// TIA Portal V19 export
FUNCTION_BLOCK "EXCHANGETRAY_ConstraintRollerCmResetOperator"   // FB51, LAD
TITLE = description
// REGION BLOCK INFO HEADER
//     //===============================================================================
//     // (company)/ (c)Copyright (year)
//     //-------------------------------------------------------------------------------
//     // Title:          cm复位操作
//     // Comment/Function:复位各cm的command信号
//     // Library/Family:   (that the source is dedicated to)
//     // Author:           (sup / zhang shilong / contact)
//     // Tested with:      (test system with FW version)
//     // Engineering:      --
//     // Restrictions:     --
//     // Requirements:     --
//     //-------------------------------------------------------------------------------
//     // Change log table:
//     // Version  | Date       | Expert in charge        | Changes applied
//     //----------|------------|-------------------------|-----------------------------
//     // 01.00.00 | dd.mm.yyyy | (name of expert)        | First released version
//     //===============================================================================
// END_REGION BLOCK INFO HEADER
// stored: MemoryReserve 100, Namespace Unit2.EM4, SetENOAutomatically false
   VAR
      instAxis1ResetMerge { S7_SetPoint := 'True'} : "LEXCHANGETRAY_AxisResetMerge";
      instAxis2ResetMerge { S7_SetPoint := 'True'} : "LEXCHANGETRAY_AxisResetMerge";
      instAxis3ResetMerge { S7_SetPoint := 'True'} : "LEXCHANGETRAY_AxisResetMerge";
      instCylinder4ResetMerge { S7_SetPoint := 'True'} : "LEXCHANGETRAY_CylinderResetMerge";
      instCylinder5ResetMerge { S7_SetPoint := 'True'} : "LEXCHANGETRAY_CylinderResetMerge";
      instCylinder6ResetMerge { S7_SetPoint := 'True'} : "LEXCHANGETRAY_CylinderResetMerge";
      instCylinder7ResetMerge { S7_SetPoint := 'True'} : "LEXCHANGETRAY_CylinderResetMerge";
   END_VAR
BEGIN

REGION Network 1 (SCL): CM1
    #instAxis1ResetMerge(ack:="Unit2.EmNodes".unitStatus.acknowledgeActive,
                       reset:="Unit2.EmNodes".unitStatus.state.resetting,
                       axis:="Unit2.EM4.ControlNodes".cm1AxisControl);
END_REGION

REGION Network 2 (SCL): CM2
   #instAxis2ResetMerge(ack := "Unit2.EmNodes".unitStatus.acknowledgeActive,
                        reset := "Unit2.EmNodes".unitStatus.state.resetting,
                        axis := "Unit2.EM4.ControlNodes".cm2AxisControl);
END_REGION

REGION Network 3 (SCL): CM3
   #instAxis3ResetMerge(ack := "Unit2.EmNodes".unitStatus.acknowledgeActive,
                        reset := "Unit2.EmNodes".unitStatus.state.resetting,
                        axis := "Unit2.EM4.ControlNodes".cm3AxisControl);
END_REGION

REGION Network 4 (SCL): CM4
   #instCylinder4ResetMerge(ack:="Unit2.EmNodes".unitStatus.acknowledgeActive,
                           reset:="Unit2.EmNodes".unitStatus.state.resetting,
                           cylinder:="Unit2.EM4.ControlNodes".cm4Cylinder);
END_REGION

REGION Network 5 (SCL): cm5
   #instCylinder5ResetMerge(ack := "Unit2.EmNodes".unitStatus.acknowledgeActive,
                            reset := "Unit2.EmNodes".unitStatus.state.resetting,
                            cylinder := "Unit2.EM4.ControlNodes".cm5Cylinder);
END_REGION

REGION Network 6 (SCL): cm6
   #instCylinder6ResetMerge(ack := "Unit2.EmNodes".unitStatus.acknowledgeActive,
                            reset := "Unit2.EmNodes".unitStatus.state.resetting,
                            cylinder := "Unit2.EM4.ControlNodes".cm6Cylinder);
END_REGION

REGION Network 7 (SCL): cm7
   #instCylinder7ResetMerge(ack := "Unit2.EmNodes".unitStatus.acknowledgeActive,
                            reset := "Unit2.EmNodes".unitStatus.state.resetting,
                            cylinder := "Unit2.EM4.ControlNodes".cm7Cylinder);
END_REGION

REGION Network 8: #####end
END_REGION
END_FUNCTION_BLOCK
